// TIA Portal V18 export
FUNCTION_BLOCK "HMI"   // FB20, LAD
TITLE = HMI
{ S7_Optimized_Access := 'TRUE' }
// Bonanza Elect TD Rev0
// Written By Kristopher Gimenez Feb 13,2023
// 
// This block and its associated DB are used for HMI specific actions, interlocks and visualizations.
// stored: AutoNumber false, MemoryReserve 100, SetENOAutomatically false
   VAR
      DHScreen : Array[0..4] of Int;   // Current Info of the Doghouse HMI
      HPUScreen : Array[0..4] of Int;   // Current Info Number of the HPU HMI
      ConsoleScreen : Array[0..4] of Int;   // Current Info Number of the Console HMI
      OscEnable : Bool;   // Oscillator Enable Bit. Set on HMI
      OscAllowEn : Bool;   // Allow Enable from HMI screen.
   END_VAR
   VAR RETAIN
      OscBumpAdj { S7_SetPoint := 'True'} : Real := 20.0;   // Amount the bump position will adjust if increment/decremented. Set on HMI
   END_VAR
   VAR
      OscBumpFwdInc : Bool;   // Used to increase the Fwd Bump by the adjust amount
      OscBumpFwdDec : Bool;   // Used to dec the Fwd Bump by the adjust amount
      OscBumpReactive : Bool;   // Used to trigger Reactive Bump. Always FWD
      OscBumpRevInc : Bool;   // Used to increase the RevBump by the adjust amount
      OscBumpRevDec : Bool;   // Used to dec the Rev Bump by the adjust amount
      OscBumpFwd : Bool;   // Bit used to increase the Home position
      OscBumpRev : Bool;   // Bit used to decrease the home position
   END_VAR
   VAR RETAIN
      OscBumpFwdDeg : Real;   // Amount of Degrees to Bump Forward
      OscBumpRevDeg : Real;   // Amount of Degress to Bump in Rev
   END_VAR
   VAR
      OscHoldButton : Bool;   // Bit used to change color of Button On HMI
      OscHold : Bool;   // Bit used to hold Osc at current position.
      OscBumpFwdButton : Bool;
      OscBumpRevButton : Bool;
      OscBumpFwdRevButtonEn : Bool;
      OscHomeRelDeg : Real;   // Relative Oscillator Home position in degrees.
   END_VAR
   VAR RETAIN
      OscP1FwdMinmA { S7_SetPoint := 'True'} : Real := 200.0;   // Min mA output for Osc FWD on P1
      OscP1FwdMaxmA { S7_SetPoint := 'True'} : Real := 600.0;   // Max mA output for Osc FWD on P1
      OscP1RevMinmA { S7_SetPoint := 'True'} : Real := 200.0;   // Min mA output for Osc Rev on P1
      OscP1RevMaxmA { S7_SetPoint := 'True'} : Real := 600.0;   // Max mA output for Osc Rev on P1
      OscP1HoldmA { S7_SetPoint := 'True'} : Real := 300.0;   // mA Setting to hold position while oscillating
      OscP2FwdMinmA { S7_SetPoint := 'True'} : Real := 200.0;   // Min mA output for Osc FWD on P2
      OscP2FwdMaxmA { S7_SetPoint := 'True'} : Real := 600.0;   // Max mA output for Osc FWD on P2
      OscP2RevMinmA { S7_SetPoint := 'True'} : Real := 200.0;   // Min mA output for Osc Rev on P2
      OscP2RevMaxmA { S7_SetPoint := 'True'} : Real := 600.0;   // Max mA output for Osc Rev on P2
      OscP2HoldmA { S7_SetPoint := 'True'} : Real := 300.0;   // mA Setting to hold position while oscillating
   END_VAR
   VAR
      OscPosZero : Bool;   // Bit used toset the current rotary position as zero degrees and reset Home.
   END_VAR
   VAR RETAIN
      OscSlewRiseFast { S7_SetPoint := 'True'} : Real := 100.0;   // Rising Slew Rate mA/sec for Flow, fast reaction
      OscSlewRiseSlow { S7_SetPoint := 'True'} : Real := 10.0;   // Rising Slew Rate mA/sec on Flow, slow reaction
      OscSlewFallFast { S7_SetPoint := 'True'} : Real := 100.0;   // Falling Slew Rate mA/sec for Flow, fast reaction
      OscSlewFallSlow { S7_SetPoint := 'True'} : Real := 10.0;   // Falling Slew Rate mA/sec on Flow, slow reaction
      OscSpeedTHper { S7_SetPoint := 'True'} : Real := 75.0;   // Speed threshold percent to determine fast or slow slew rates
      OscSpeedHoldper { S7_SetPoint := 'True'} : Real := 95.0;   // Speed threshold percent to where control is held.
      OscSpeedFwdRPM { S7_SetPoint := 'True'} : Real := 15.0;   // Osc FWD speed setpoint. Set on HMI
      OscSpeedRevRPM { S7_SetPoint := 'True'} : Real := 15.0;   // Osc Rev speed setpoint Set on HMI
   END_VAR
   VAR
      OscSpeedFwdZone1 : Real;   // Calc value base on Input and TH percent. Below this speed setpoint - fast ramp up to the speed
      OscSpeedFwdZone2 : Real;   // Calc value base on Input and TH percent, Between Set 1 and Set 2 - Slow ramp up to speed
      OscSpeedFwdZone3 : Real;   // Calc value base on Input and TH percent,Between Set 2 and Set 3 - Maintina Speed
      OscSpeedFwdZone4 : Real;   // Calc value base on Input and TH percent,Between Set 3 and 4 - Slow Ramp Down. Above this speed Fast ramp down
      OscSpeedRevZone1 : Real;   // Calc value base on Input and TH percent. Below this speed setpoint - fast ramp up to the speed
      OscSpeedRevZone2 : Real;   // Calc value base on Input and TH percent, Between Set 1 and Set 2 - Slow ramp up to speed
      OscSpeedRevZone3 : Real;   // Calc value base on Input and TH percent,Between Set 2 and Set 3 - Maintina Speed
      OscSpeedRevZone4 : Real;   // Calc value base on Input and TH percent,Between Set 3 and 4 - Slow Ramp Down. Above this speed Fast ramp down
      OscStart : Bool;   // Bit used to start Oscillating
      OscStartButton : Bool;   // Bit used to change color of Button On HMI
      OscStop : Bool;   // Bit used to Stop Oscillating or Holding
      OscStopButton : Bool;   // Bit used to change color of Button On HMI
   END_VAR
   VAR RETAIN
      OscTorqAdj { S7_SetPoint := 'True'} : Real := 500.0;   // Amount the torq will adjust if increment/decremented. Set on HMI
      OscTorqFwdFtLbs : Real := 5000.0;   // Osc fwd torq setpoint
   END_VAR
   VAR
      OscTorqFwdInc : Bool;   // Increment Torq Fwd
      OscTorqFwdDec : Bool;   // Decrement Torq Fwd
      OscTorqRevInc : Bool;   // Increment Torq Rev
   END_VAR
   VAR RETAIN
      OscTorqRevFtLbs : Real := 5000.0;   // Osc Rev Torq Setpoint
   END_VAR
   VAR
      OscTorqRevDec : Bool;   // Decrement Torq REv
      OscTorqSetPSI : Real;
   END_VAR
   VAR RETAIN
      OscTurnAdj { S7_SetPoint := 'True'} : Real := 0.25;   // Amount the turns will adjust if increment/decremented. Set on HMI
      OscTurnFwd : Real := 1.0;   // Osc Fwd Turns
   END_VAR
   VAR
      OscTurnFwdInc : Bool;   // Increment Turns Fwd
      OscTurnFwdDec : Bool;   // Decrement Turns Fwd
   END_VAR
   VAR RETAIN
      OscTurnRev : Real := 1.0;   // Osc Rev Turns
   END_VAR
   VAR
      OscTurnRevInc : Bool;   // Increment Turns Rev
      OscTurnRevDec : Bool;   // Decrement Turns Rev
      OscTorqFwdLowLimFtlbs : Real;   // Forward torq lower limit based on input and settings
      OscTorqFwdHighLimFtLbs : Real;   // Forward torq high limit based on input and settings
      OscTorqRevLowLimFtlbs : Real;   // Reverse torq lower limit based on input and settings
      OscTorqRevHighLimFtLbs : Real;   // Reverse torq high limit based on input and settings
      OscHomeLowRelDeg : Real;   // Rel Home Position minus 1 count range
      OscHomeLow2RelDeg : Real;   // Rel Home Position minus 2 count range
      OscHomeHighRelDeg : Real;   // Rel Home Position plus 1 count range
      OscHomeHigh2RelDeg : Real;   // Rel Home Position plus 2 count range
      OscPosDeg : Real;   // Degrees of from Home position
      SpareVolts : Real := 0.0;   // Dummy spare Output value used for display
      Spare4MA : Real := 4.0;   // Dummy spare Output value 4ma
      LampTest : Bool;   // Bit used to trigger Console lamp test from HMI
      LampTestLamp_TP { S7_SetPoint := 'True'} : TP_TIME;
      LampTestHorn_TP { S7_SetPoint := 'True'} : TP_TIME;
      ScreenNameInvis { S7_SetPoint := 'True'} : Bool;   // Used to Turn off Screen Name
      ScreenBypassVis : Bool;
      ScreenLampTestVis : Bool;
      HornSilence_TOF { S7_SetPoint := 'True'} : TOF_TIME;
      HornSilenceReset { S7_SetPoint := 'True'} : Bool;   // Horn Silence Bit set on HMI
      Alarms1 : Int;
      Alarms2 : Int;
      Warnings1 : Int;
      Alarms1_To_Unified : Array[0..15] of Bool;
      Alarms2_To_Unified : Array[0..15] of Bool;
      Warnings1_To_Unified : Array[0..15] of Bool;
   END_VAR
   VAR_TEMP
      TempReal : Real;
   END_VAR
   VAR_TEMP   // added for the SCL form of the ladder/FBD networks
      _w1 : Bool;
   END_VAR
BEGIN

REGION Network 1: Oscillator Enable
   // Allow Enable Osciallor Set from HMI if  in Drill, throttle pot set to min and TD stopped, low speed. 
   // HMI Used to Set Enable
   // Reset if Interlocks not met
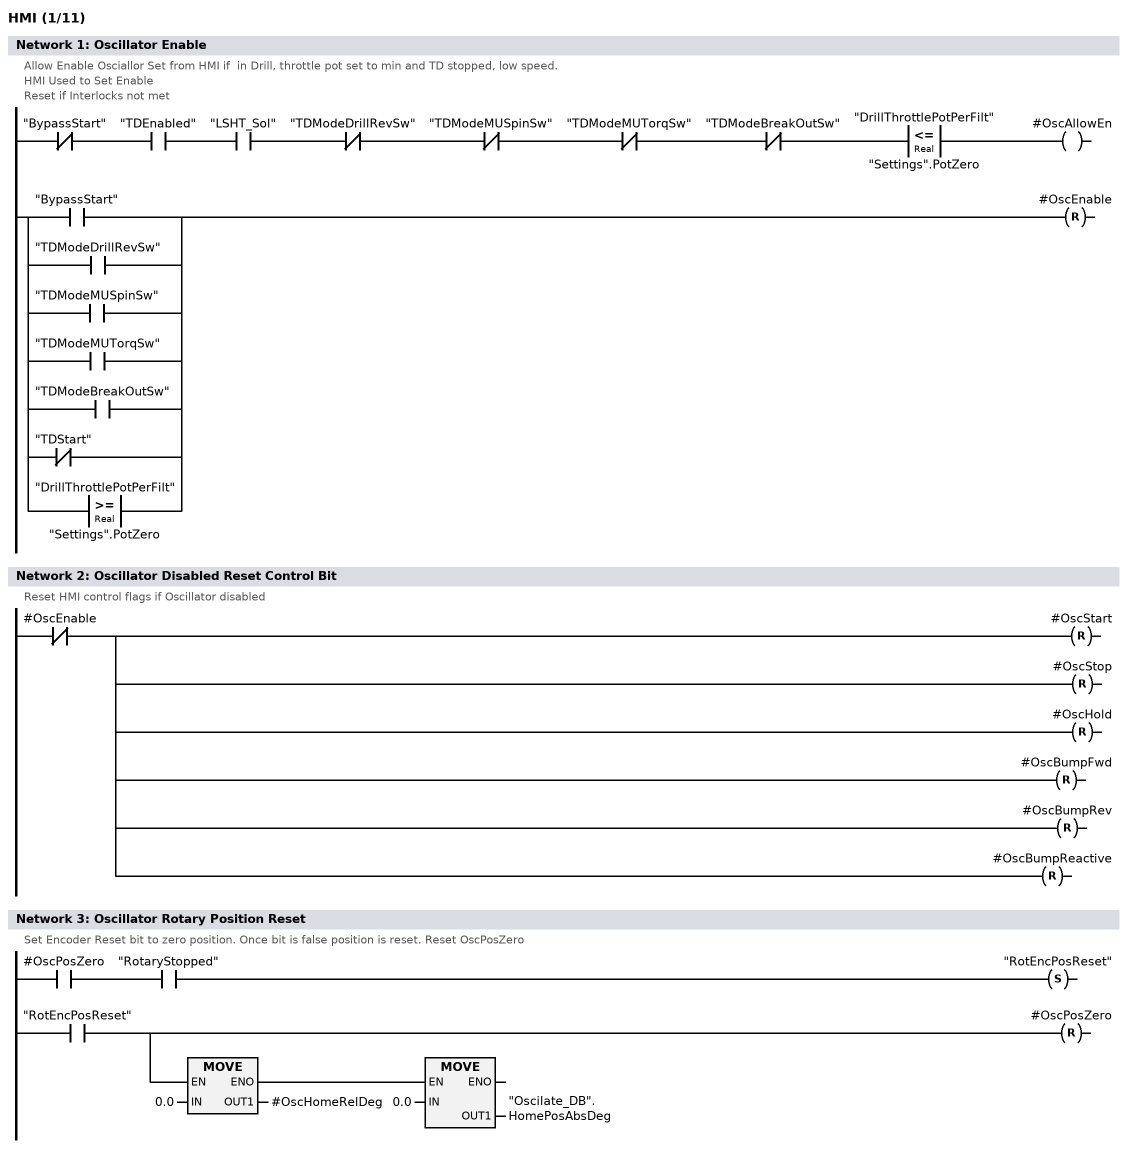
   RUNG wire#powerrail
      I_Contact( "BypassStart" )
      Contact( "TDEnabled" )
      Contact( "LSHT_Sol" )
      I_Contact( "TDModeDrillRevSw" )
      I_Contact( "TDModeMUSpinSw" )
      I_Contact( "TDModeMUTorqSw" )
      I_Contact( "TDModeBreakOutSw" )
      { S7_Templates := "SrcType := Real" } LE_Contact(in1 := "DrillThrottlePotPerFilt", in2 := "Settings".PotZero)
      Coil( #OscAllowEn )
   END_RUNG
   RUNG wire#powerrail
      Contact( "BypassStart" )
      wire#w1
      R_Coil( #OscEnable )
   END_RUNG
   RUNG wire#powerrail
      Contact( "TDModeDrillRevSw" )
   END_RUNG wire#w1
   RUNG wire#powerrail
      Contact( "TDModeMUSpinSw" )
   END_RUNG wire#w1
   RUNG wire#powerrail
      Contact( "TDModeMUTorqSw" )
   END_RUNG wire#w1
   RUNG wire#powerrail
      Contact( "TDModeBreakOutSw" )
   END_RUNG wire#w1
   RUNG wire#powerrail
      I_Contact( "TDStart" )
   END_RUNG wire#w1
   RUNG wire#powerrail
      { S7_Templates := "SrcType := Real" } GE_Contact(in1 := "DrillThrottlePotPerFilt", in2 := "Settings".PotZero)
   END_RUNG wire#w1
   // the same network as SCL:
   #OscAllowEn := NOT "BypassStart" AND "TDEnabled" AND "LSHT_Sol" AND NOT "TDModeDrillRevSw" AND NOT "TDModeMUSpinSw" AND NOT "TDModeMUTorqSw" AND NOT "TDModeBreakOutSw" AND ("DrillThrottlePotPerFilt" <= "Settings".PotZero);
   IF "BypassStart" OR "TDModeDrillRevSw" OR "TDModeMUSpinSw" OR "TDModeMUTorqSw" OR "TDModeBreakOutSw" OR NOT "TDStart" OR ("DrillThrottlePotPerFilt" >= "Settings".PotZero) THEN
       #OscEnable := FALSE;
   END_IF;
END_REGION

REGION Network 2: Oscillator Disabled Reset Control Bit
   // Reset HMI control flags if Oscillator disabled
   RUNG wire#powerrail
      I_Contact( #OscEnable )
      wire#w1
      R_Coil( #OscStart )
   END_RUNG
   RUNG wire#w1
      R_Coil( #OscStop )
   END_RUNG
   RUNG wire#w1
      R_Coil( #OscHold )
   END_RUNG
   RUNG wire#w1
      R_Coil( #OscBumpFwd )
   END_RUNG
   RUNG wire#w1
      R_Coil( #OscBumpRev )
   END_RUNG
   RUNG wire#w1
      R_Coil( #OscBumpReactive )
   END_RUNG
   // the same network as SCL:
   IF NOT #OscEnable THEN
       #OscStart := FALSE;
       #OscStop := FALSE;
       #OscHold := FALSE;
       #OscBumpFwd := FALSE;
       #OscBumpRev := FALSE;
       #OscBumpReactive := FALSE;
   END_IF;
END_REGION

REGION Network 3: Oscillator Rotary Position Reset
   // Set Encoder Reset bit to zero position. Once bit is false position is reset. Reset OscPosZero
   RUNG wire#powerrail
      Contact( #OscPosZero )
      Contact( "RotaryStopped" )
      S_Coil( "RotEncPosReset" )
   END_RUNG
   RUNG wire#powerrail
      Contact( "RotEncPosReset" )
      wire#w1
      R_Coil( #OscPosZero )
   END_RUNG
   RUNG wire#w1
      Move(in := 0.0, out1 => #OscHomeRelDeg)
      Move(in := 0.0, out1 => "Oscilate_DB".HomePosAbsDeg)
   END_RUNG
   // the same network as SCL:
   IF #OscPosZero AND "RotaryStopped" THEN "RotEncPosReset" := TRUE; END_IF;
   IF "RotEncPosReset" THEN
       #OscPosZero := FALSE;
       #OscHomeRelDeg := 0.0;
       "Oscilate_DB".HomePosAbsDeg := 0.0;
   END_IF;
END_REGION

REGION Network 4: Oscillator Position
   // Determine Oscillation position based on home position and actual absolute position
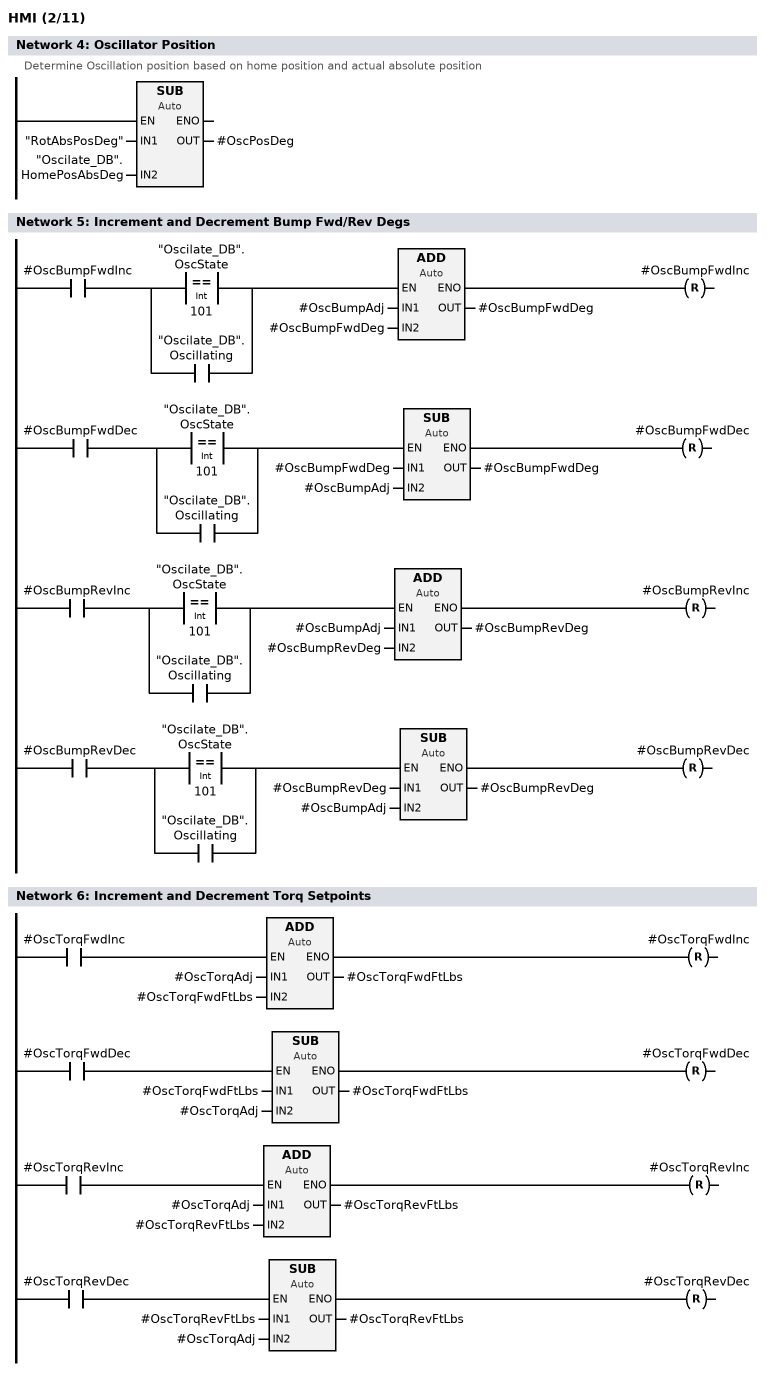
   RUNG wire#powerrail
      Sub(in1 := "RotAbsPosDeg", in2 := "Oscilate_DB".HomePosAbsDeg, out => #OscPosDeg)
   END_RUNG
   // the same network as SCL:
   #OscPosDeg := "RotAbsPosDeg" - "Oscilate_DB".HomePosAbsDeg;
END_REGION

REGION Network 5: Increment and Decrement Bump Fwd/Rev Degs
   RUNG wire#powerrail
      Contact( #OscBumpFwdInc )
      wire#w1
      { S7_Templates := "SrcType := Int" } EQ_Contact(in1 := "Oscilate_DB".OscState, in2 := 101)
      wire#w2
      Add(in1 := #OscBumpAdj, in2 := #OscBumpFwdDeg, out => #OscBumpFwdDeg)
      R_Coil( #OscBumpFwdInc )
   END_RUNG
   RUNG wire#w1
      Contact( "Oscilate_DB".Oscillating )
   END_RUNG wire#w2
   RUNG wire#powerrail
      Contact( #OscBumpFwdDec )
      wire#w3
      { S7_Templates := "SrcType := Int" } EQ_Contact(in1 := "Oscilate_DB".OscState, in2 := 101)
      wire#w4
      Sub(in1 := #OscBumpFwdDeg, in2 := #OscBumpAdj, out => #OscBumpFwdDeg)
      R_Coil( #OscBumpFwdDec )
   END_RUNG
   RUNG wire#w3
      Contact( "Oscilate_DB".Oscillating )
   END_RUNG wire#w4
   RUNG wire#powerrail
      Contact( #OscBumpRevInc )
      wire#w5
      { S7_Templates := "SrcType := Int" } EQ_Contact(in1 := "Oscilate_DB".OscState, in2 := 101)
      wire#w6
      Add(in1 := #OscBumpAdj, in2 := #OscBumpRevDeg, out => #OscBumpRevDeg)
      R_Coil( #OscBumpRevInc )
   END_RUNG
   RUNG wire#w5
      Contact( "Oscilate_DB".Oscillating )
   END_RUNG wire#w6
   RUNG wire#powerrail
      Contact( #OscBumpRevDec )
      wire#w7
      { S7_Templates := "SrcType := Int" } EQ_Contact(in1 := "Oscilate_DB".OscState, in2 := 101)
      wire#w8
      Sub(in1 := #OscBumpRevDeg, in2 := #OscBumpAdj, out => #OscBumpRevDeg)
      R_Coil( #OscBumpRevDec )
   END_RUNG
   RUNG wire#w7
      Contact( "Oscilate_DB".Oscillating )
   END_RUNG wire#w8
   // the same network as SCL:
   IF #OscBumpFwdInc AND (("Oscilate_DB".OscState = 101) OR "Oscilate_DB".Oscillating) THEN
       #OscBumpFwdDeg := #OscBumpAdj + #OscBumpFwdDeg;
       #OscBumpFwdInc := FALSE;
   END_IF;
   IF #OscBumpFwdDec AND (("Oscilate_DB".OscState = 101) OR "Oscilate_DB".Oscillating) THEN
       #OscBumpFwdDeg := #OscBumpFwdDeg - #OscBumpAdj;
       #OscBumpFwdDec := FALSE;
   END_IF;
   IF #OscBumpRevInc AND (("Oscilate_DB".OscState = 101) OR "Oscilate_DB".Oscillating) THEN
       #OscBumpRevDeg := #OscBumpAdj + #OscBumpRevDeg;
       #OscBumpRevInc := FALSE;
   END_IF;
   IF #OscBumpRevDec AND (("Oscilate_DB".OscState = 101) OR "Oscilate_DB".Oscillating) THEN
       #OscBumpRevDeg := #OscBumpRevDeg - #OscBumpAdj;
       #OscBumpRevDec := FALSE;
   END_IF;
END_REGION

REGION Network 6: Increment and Decrement Torq Setpoints
   RUNG wire#powerrail
      Contact( #OscTorqFwdInc )
      Add(in1 := #OscTorqAdj, in2 := #OscTorqFwdFtLbs, out => #OscTorqFwdFtLbs)
      R_Coil( #OscTorqFwdInc )
   END_RUNG
   RUNG wire#powerrail
      Contact( #OscTorqFwdDec )
      Sub(in1 := #OscTorqFwdFtLbs, in2 := #OscTorqAdj, out => #OscTorqFwdFtLbs)
      R_Coil( #OscTorqFwdDec )
   END_RUNG
   RUNG wire#powerrail
      Contact( #OscTorqRevInc )
      Add(in1 := #OscTorqAdj, in2 := #OscTorqRevFtLbs, out => #OscTorqRevFtLbs)
      R_Coil( #OscTorqRevInc )
   END_RUNG
   RUNG wire#powerrail
      Contact( #OscTorqRevDec )
      Sub(in1 := #OscTorqRevFtLbs, in2 := #OscTorqAdj, out => #OscTorqRevFtLbs)
      R_Coil( #OscTorqRevDec )
   END_RUNG
   // the same network as SCL:
   IF #OscTorqFwdInc THEN
       #OscTorqFwdFtLbs := #OscTorqAdj + #OscTorqFwdFtLbs;
       #OscTorqFwdInc := FALSE;
   END_IF;
   IF #OscTorqFwdDec THEN
       #OscTorqFwdFtLbs := #OscTorqFwdFtLbs - #OscTorqAdj;
       #OscTorqFwdDec := FALSE;
   END_IF;
   IF #OscTorqRevInc THEN
       #OscTorqRevFtLbs := #OscTorqAdj + #OscTorqRevFtLbs;
       #OscTorqRevInc := FALSE;
   END_IF;
   IF #OscTorqRevDec THEN
       #OscTorqRevFtLbs := #OscTorqRevFtLbs - #OscTorqAdj;
       #OscTorqRevDec := FALSE;
   END_IF;
END_REGION

REGION Network 7: Increment and Decrement Turns
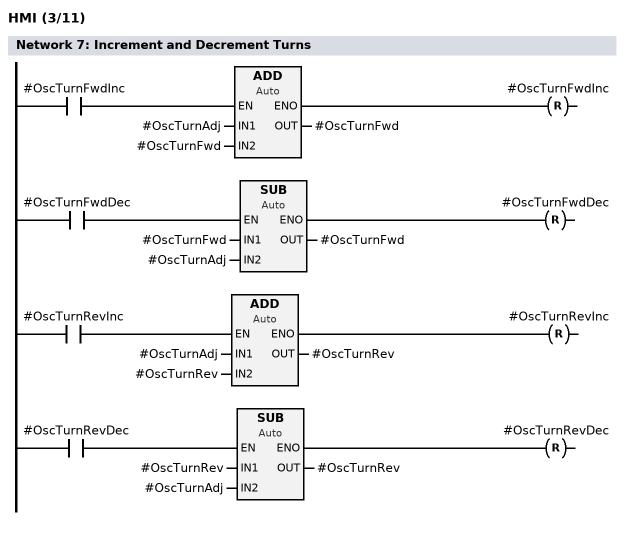
   RUNG wire#powerrail
      Contact( #OscTurnFwdInc )
      Add(in1 := #OscTurnAdj, in2 := #OscTurnFwd, out => #OscTurnFwd)
      R_Coil( #OscTurnFwdInc )
   END_RUNG
   RUNG wire#powerrail
      Contact( #OscTurnFwdDec )
      Sub(in1 := #OscTurnFwd, in2 := #OscTurnAdj, out => #OscTurnFwd)
      R_Coil( #OscTurnFwdDec )
   END_RUNG
   RUNG wire#powerrail
      Contact( #OscTurnRevInc )
      Add(in1 := #OscTurnAdj, in2 := #OscTurnRev, out => #OscTurnRev)
      R_Coil( #OscTurnRevInc )
   END_RUNG
   RUNG wire#powerrail
      Contact( #OscTurnRevDec )
      Sub(in1 := #OscTurnRev, in2 := #OscTurnAdj, out => #OscTurnRev)
      R_Coil( #OscTurnRevDec )
   END_RUNG
   // the same network as SCL:
   IF #OscTurnFwdInc THEN
       #OscTurnFwd := #OscTurnAdj + #OscTurnFwd;
       #OscTurnFwdInc := FALSE;
   END_IF;
   IF #OscTurnFwdDec THEN
       #OscTurnFwd := #OscTurnFwd - #OscTurnAdj;
       #OscTurnFwdDec := FALSE;
   END_IF;
   IF #OscTurnRevInc THEN
       #OscTurnRev := #OscTurnAdj + #OscTurnRev;
       #OscTurnRevInc := FALSE;
   END_IF;
   IF #OscTurnRevDec THEN
       #OscTurnRev := #OscTurnRev - #OscTurnAdj;
       #OscTurnRevDec := FALSE;
   END_IF;
END_REGION

REGION Network 8: Oscillator Input Limits Checks
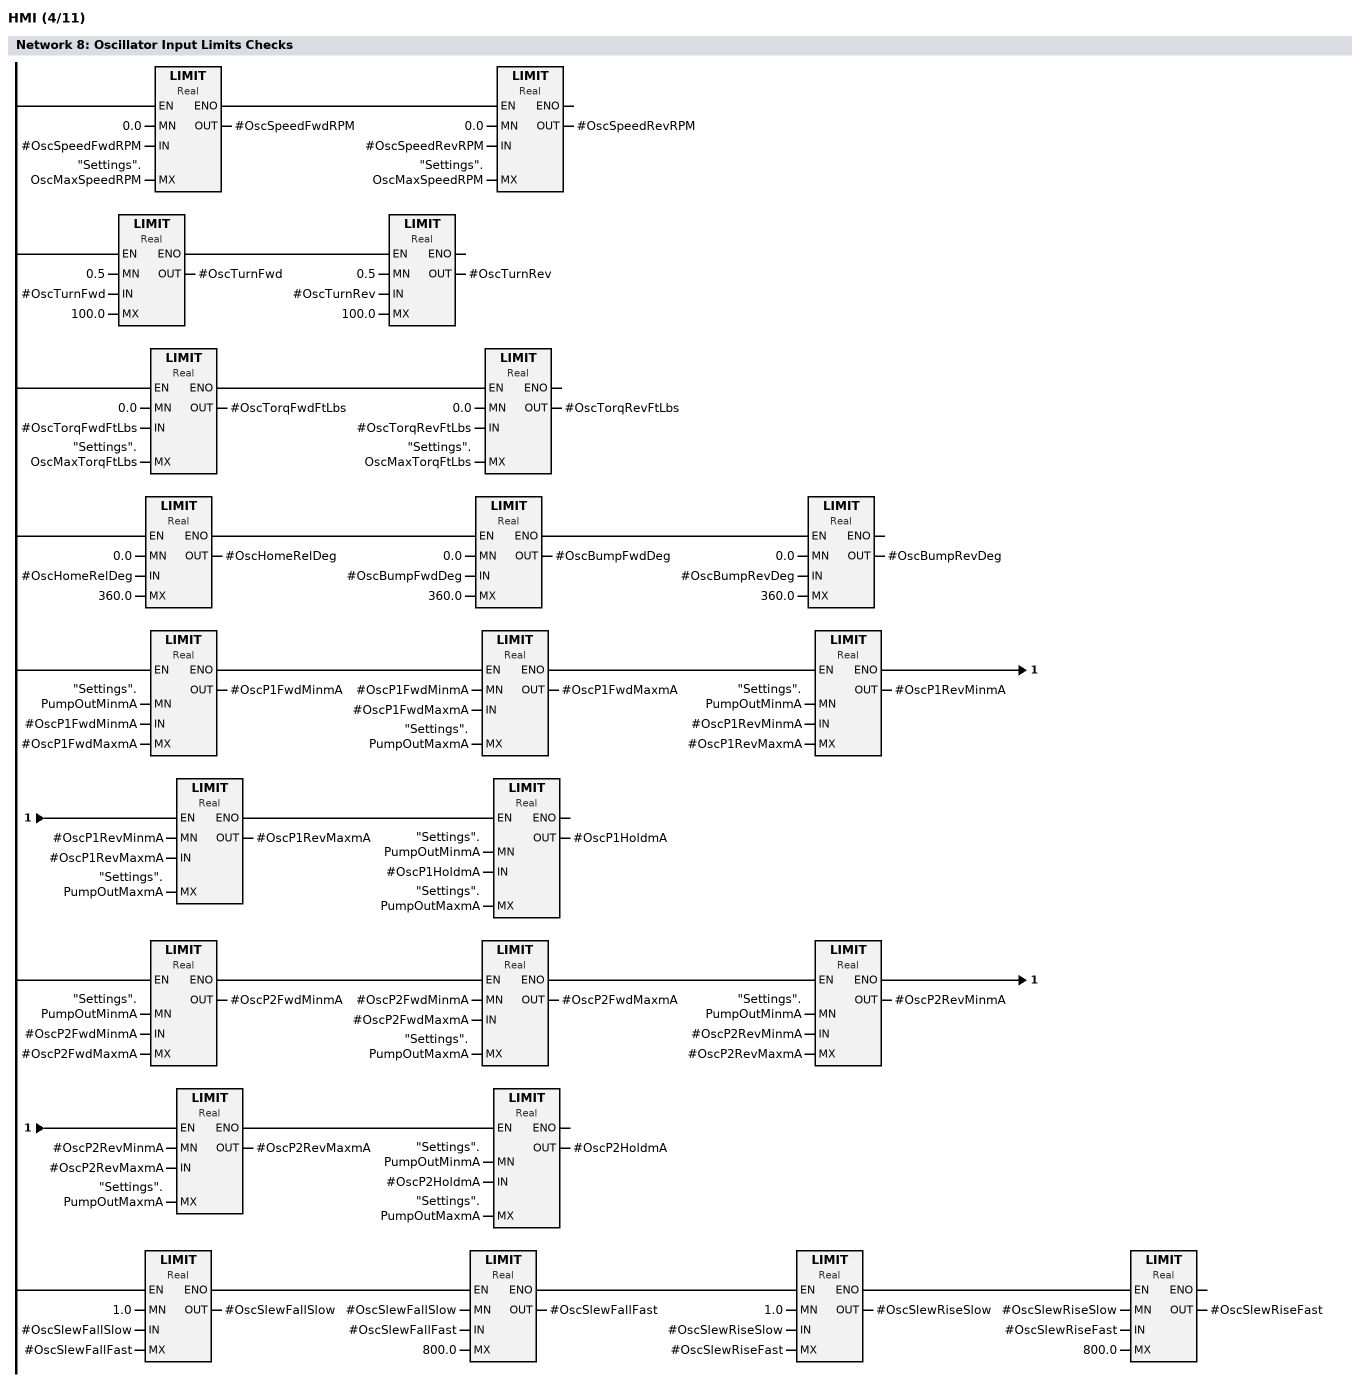
   RUNG wire#powerrail
      { S7_Templates := "value_type := Real" } Limit(mn := 0.0, in := #OscSpeedFwdRPM, mx := "Settings".OscMaxSpeedRPM, out => #OscSpeedFwdRPM)
      { S7_Templates := "value_type := Real" } Limit(mn := 0.0, in := #OscSpeedRevRPM, mx := "Settings".OscMaxSpeedRPM, out => #OscSpeedRevRPM)
   END_RUNG
   RUNG wire#powerrail
      { S7_Templates := "value_type := Real" } Limit(mn := 0.5, in := #OscTurnFwd, mx := 100.0, out => #OscTurnFwd)
      { S7_Templates := "value_type := Real" } Limit(mn := 0.5, in := #OscTurnRev, mx := 100.0, out => #OscTurnRev)
   END_RUNG
   RUNG wire#powerrail
      { S7_Templates := "value_type := Real" } Limit(mn := 0.0, in := #OscTorqFwdFtLbs, mx := "Settings".OscMaxTorqFtLbs, out => #OscTorqFwdFtLbs)
      { S7_Templates := "value_type := Real" } Limit(mn := 0.0, in := #OscTorqRevFtLbs, mx := "Settings".OscMaxTorqFtLbs, out => #OscTorqRevFtLbs)
   END_RUNG
   RUNG wire#powerrail
      { S7_Templates := "value_type := Real" } Limit(mn := 0.0, in := #OscHomeRelDeg, mx := 360.0, out => #OscHomeRelDeg)
      { S7_Templates := "value_type := Real" } Limit(mn := 0.0, in := #OscBumpFwdDeg, mx := 360.0, out => #OscBumpFwdDeg)
      { S7_Templates := "value_type := Real" } Limit(mn := 0.0, in := #OscBumpRevDeg, mx := 360.0, out => #OscBumpRevDeg)
   END_RUNG
   RUNG wire#powerrail
      { S7_Templates := "value_type := Real" } Limit(mn := "Settings".PumpOutMinmA, in := #OscP1FwdMinmA, mx := #OscP1FwdMaxmA, out => #OscP1FwdMinmA)
      { S7_Templates := "value_type := Real" } Limit(mn := #OscP1FwdMinmA, in := #OscP1FwdMaxmA, mx := "Settings".PumpOutMaxmA, out => #OscP1FwdMaxmA)
      { S7_Templates := "value_type := Real" } Limit(mn := "Settings".PumpOutMinmA, in := #OscP1RevMinmA, mx := #OscP1RevMaxmA, out => #OscP1RevMinmA)
      { S7_Templates := "value_type := Real" } Limit(mn := #OscP1RevMinmA, in := #OscP1RevMaxmA, mx := "Settings".PumpOutMaxmA, out => #OscP1RevMaxmA)
      { S7_Templates := "value_type := Real" } Limit(mn := "Settings".PumpOutMinmA, in := #OscP1HoldmA, mx := "Settings".PumpOutMaxmA, out => #OscP1HoldmA)
   END_RUNG
   RUNG wire#powerrail
      { S7_Templates := "value_type := Real" } Limit(mn := "Settings".PumpOutMinmA, in := #OscP2FwdMinmA, mx := #OscP2FwdMaxmA, out => #OscP2FwdMinmA)
      { S7_Templates := "value_type := Real" } Limit(mn := #OscP2FwdMinmA, in := #OscP2FwdMaxmA, mx := "Settings".PumpOutMaxmA, out => #OscP2FwdMaxmA)
      { S7_Templates := "value_type := Real" } Limit(mn := "Settings".PumpOutMinmA, in := #OscP2RevMinmA, mx := #OscP2RevMaxmA, out => #OscP2RevMinmA)
      { S7_Templates := "value_type := Real" } Limit(mn := #OscP2RevMinmA, in := #OscP2RevMaxmA, mx := "Settings".PumpOutMaxmA, out => #OscP2RevMaxmA)
      { S7_Templates := "value_type := Real" } Limit(mn := "Settings".PumpOutMinmA, in := #OscP2HoldmA, mx := "Settings".PumpOutMaxmA, out => #OscP2HoldmA)
   END_RUNG
   RUNG wire#powerrail
      { S7_Templates := "value_type := Real" } Limit(mn := 1.0, in := #OscSlewFallSlow, mx := #OscSlewFallFast, out => #OscSlewFallSlow)
      { S7_Templates := "value_type := Real" } Limit(mn := #OscSlewFallSlow, in := #OscSlewFallFast, mx := 800.0, out => #OscSlewFallFast)
      { S7_Templates := "value_type := Real" } Limit(mn := 1.0, in := #OscSlewRiseSlow, mx := #OscSlewRiseFast, out => #OscSlewRiseSlow)
      { S7_Templates := "value_type := Real" } Limit(mn := #OscSlewRiseSlow, in := #OscSlewRiseFast, mx := 800.0, out => #OscSlewRiseFast)
   END_RUNG
   // the same network as SCL:
   #OscSpeedFwdRPM := LIMIT(MN := 0.0, IN := #OscSpeedFwdRPM, MX := "Settings".OscMaxSpeedRPM);
   #OscSpeedRevRPM := LIMIT(MN := 0.0, IN := #OscSpeedRevRPM, MX := "Settings".OscMaxSpeedRPM);
   #OscTurnFwd := LIMIT(MN := 0.5, IN := #OscTurnFwd, MX := 100.0);
   #OscTurnRev := LIMIT(MN := 0.5, IN := #OscTurnRev, MX := 100.0);
   #OscTorqFwdFtLbs := LIMIT(MN := 0.0, IN := #OscTorqFwdFtLbs, MX := "Settings".OscMaxTorqFtLbs);
   #OscTorqRevFtLbs := LIMIT(MN := 0.0, IN := #OscTorqRevFtLbs, MX := "Settings".OscMaxTorqFtLbs);
   #OscHomeRelDeg := LIMIT(MN := 0.0, IN := #OscHomeRelDeg, MX := 360.0);
   #OscBumpFwdDeg := LIMIT(MN := 0.0, IN := #OscBumpFwdDeg, MX := 360.0);
   #OscBumpRevDeg := LIMIT(MN := 0.0, IN := #OscBumpRevDeg, MX := 360.0);
   #OscP1FwdMinmA := LIMIT(MN := "Settings".PumpOutMinmA, IN := #OscP1FwdMinmA, MX := #OscP1FwdMaxmA);
   #OscP1FwdMaxmA := LIMIT(MN := #OscP1FwdMinmA, IN := #OscP1FwdMaxmA, MX := "Settings".PumpOutMaxmA);
   #OscP1RevMinmA := LIMIT(MN := "Settings".PumpOutMinmA, IN := #OscP1RevMinmA, MX := #OscP1RevMaxmA);
   #OscP1RevMaxmA := LIMIT(MN := #OscP1RevMinmA, IN := #OscP1RevMaxmA, MX := "Settings".PumpOutMaxmA);
   #OscP1HoldmA := LIMIT(MN := "Settings".PumpOutMinmA, IN := #OscP1HoldmA, MX := "Settings".PumpOutMaxmA);
   #OscP2FwdMinmA := LIMIT(MN := "Settings".PumpOutMinmA, IN := #OscP2FwdMinmA, MX := #OscP2FwdMaxmA);
   #OscP2FwdMaxmA := LIMIT(MN := #OscP2FwdMinmA, IN := #OscP2FwdMaxmA, MX := "Settings".PumpOutMaxmA);
   #OscP2RevMinmA := LIMIT(MN := "Settings".PumpOutMinmA, IN := #OscP2RevMinmA, MX := #OscP2RevMaxmA);
   #OscP2RevMaxmA := LIMIT(MN := #OscP2RevMinmA, IN := #OscP2RevMaxmA, MX := "Settings".PumpOutMaxmA);
   #OscP2HoldmA := LIMIT(MN := "Settings".PumpOutMinmA, IN := #OscP2HoldmA, MX := "Settings".PumpOutMaxmA);
   #OscSlewFallSlow := LIMIT(MN := 1.0, IN := #OscSlewFallSlow, MX := #OscSlewFallFast);
   #OscSlewFallFast := LIMIT(MN := #OscSlewFallSlow, IN := #OscSlewFallFast, MX := 800.0);
   #OscSlewRiseSlow := LIMIT(MN := 1.0, IN := #OscSlewRiseSlow, MX := #OscSlewRiseFast);
   #OscSlewRiseFast := LIMIT(MN := #OscSlewRiseSlow, IN := #OscSlewRiseFast, MX := 800.0);
END_REGION

REGION Network 9: Calculate Torq Setpoint
   // Only Fwd Torq is used to set torq
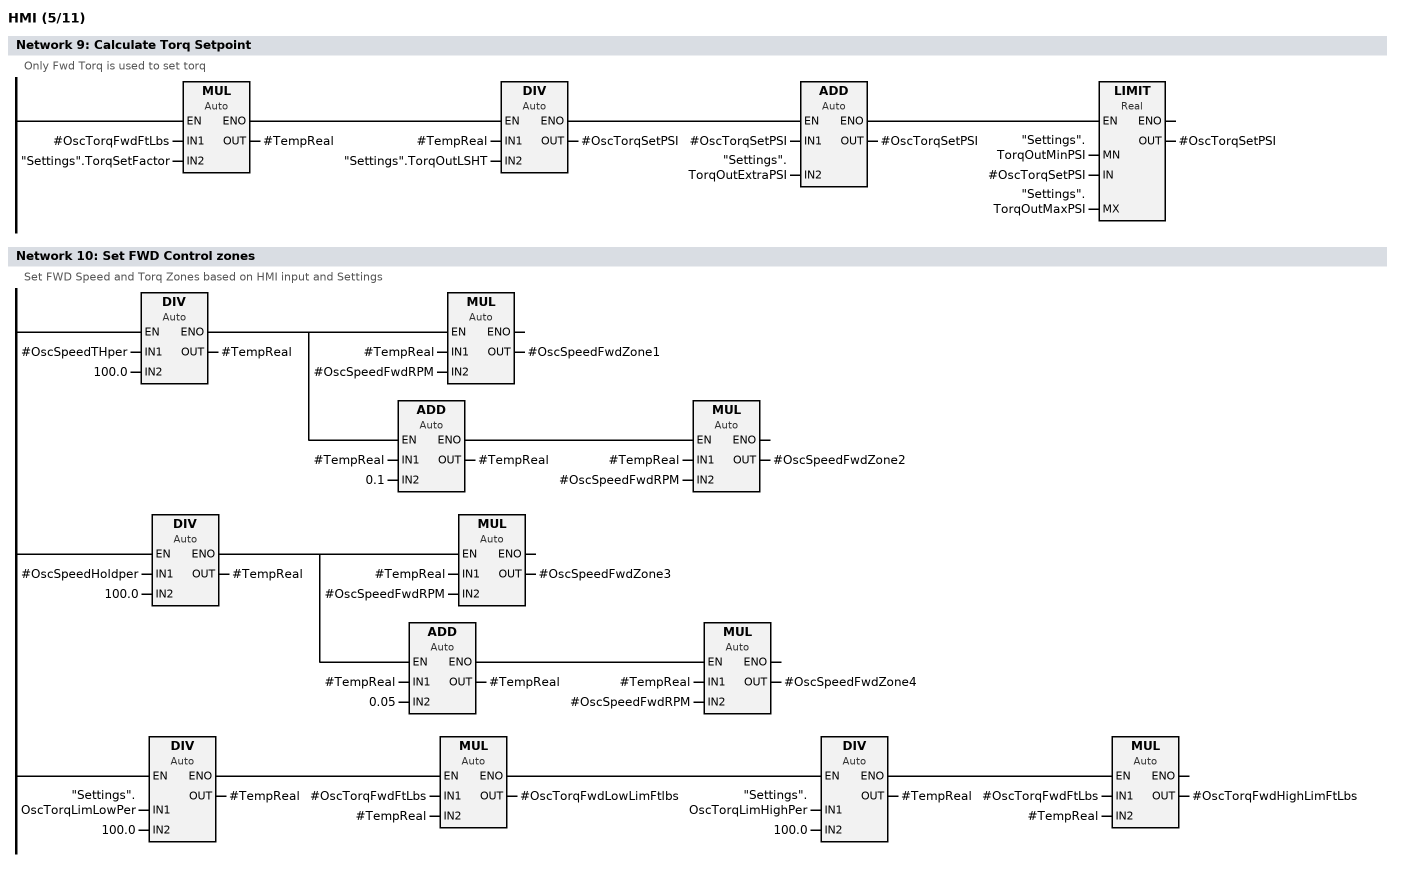
   RUNG wire#powerrail
      Mul(in1 := #OscTorqFwdFtLbs, in2 := "Settings".TorqSetFactor, out => #TempReal)
      Div(in1 := #TempReal, in2 := "Settings".TorqOutLSHT, out => #OscTorqSetPSI)
      Add(in1 := #OscTorqSetPSI, in2 := "Settings".TorqOutExtraPSI, out => #OscTorqSetPSI)
      { S7_Templates := "value_type := Real" } Limit(mn := "Settings".TorqOutMinPSI, in := #OscTorqSetPSI, mx := "Settings".TorqOutMaxPSI, out => #OscTorqSetPSI)
   END_RUNG
   // the same network as SCL:
   #TempReal := #OscTorqFwdFtLbs * "Settings".TorqSetFactor;
   #OscTorqSetPSI := #TempReal / "Settings".TorqOutLSHT;
   #OscTorqSetPSI := #OscTorqSetPSI + "Settings".TorqOutExtraPSI;
   #OscTorqSetPSI := LIMIT(MN := "Settings".TorqOutMinPSI, IN := #OscTorqSetPSI, MX := "Settings".TorqOutMaxPSI);
END_REGION

REGION Network 10: Set FWD Control zones
   // Set FWD Speed and Torq Zones based on HMI input and Settings
   RUNG wire#powerrail
      Div(in1 := #OscSpeedTHper, in2 := 100.0, out => #TempReal)
      wire#w1
      Mul(in1 := #TempReal, in2 := #OscSpeedFwdRPM, out => #OscSpeedFwdZone1)
   END_RUNG
   RUNG wire#w1
      Add(in1 := #TempReal, in2 := 0.1, out => #TempReal)
      Mul(in1 := #TempReal, in2 := #OscSpeedFwdRPM, out => #OscSpeedFwdZone2)
   END_RUNG
   RUNG wire#powerrail
      Div(in1 := #OscSpeedHoldper, in2 := 100.0, out => #TempReal)
      wire#w2
      Mul(in1 := #TempReal, in2 := #OscSpeedFwdRPM, out => #OscSpeedFwdZone3)
   END_RUNG
   RUNG wire#w2
      Add(in1 := #TempReal, in2 := 0.05, out => #TempReal)
      Mul(in1 := #TempReal, in2 := #OscSpeedFwdRPM, out => #OscSpeedFwdZone4)
   END_RUNG
   RUNG wire#powerrail
      Div(in1 := "Settings".OscTorqLimLowPer, in2 := 100.0, out => #TempReal)
      Mul(in1 := #OscTorqFwdFtLbs, in2 := #TempReal, out => #OscTorqFwdLowLimFtlbs)
      Div(in1 := "Settings".OscTorqLimHighPer, in2 := 100.0, out => #TempReal)
      Mul(in1 := #OscTorqFwdFtLbs, in2 := #TempReal, out => #OscTorqFwdHighLimFtLbs)
   END_RUNG
   // the same network as SCL:
   #TempReal := #OscSpeedTHper / 100.0;
   #OscSpeedFwdZone1 := #TempReal * #OscSpeedFwdRPM;
   #TempReal := #TempReal + 0.1;
   #OscSpeedFwdZone2 := #TempReal * #OscSpeedFwdRPM;
   #TempReal := #OscSpeedHoldper / 100.0;
   #OscSpeedFwdZone3 := #TempReal * #OscSpeedFwdRPM;
   #TempReal := #TempReal + 0.05;
   #OscSpeedFwdZone4 := #TempReal * #OscSpeedFwdRPM;
   #TempReal := "Settings".OscTorqLimLowPer / 100.0;
   #OscTorqFwdLowLimFtlbs := #OscTorqFwdFtLbs * #TempReal;
   #TempReal := "Settings".OscTorqLimHighPer / 100.0;
   #OscTorqFwdHighLimFtLbs := #OscTorqFwdFtLbs * #TempReal;
END_REGION

REGION Network 11: Set Rev Controls zones
   // Set Rev Speed and Torq Zones based on HMI input and Settings
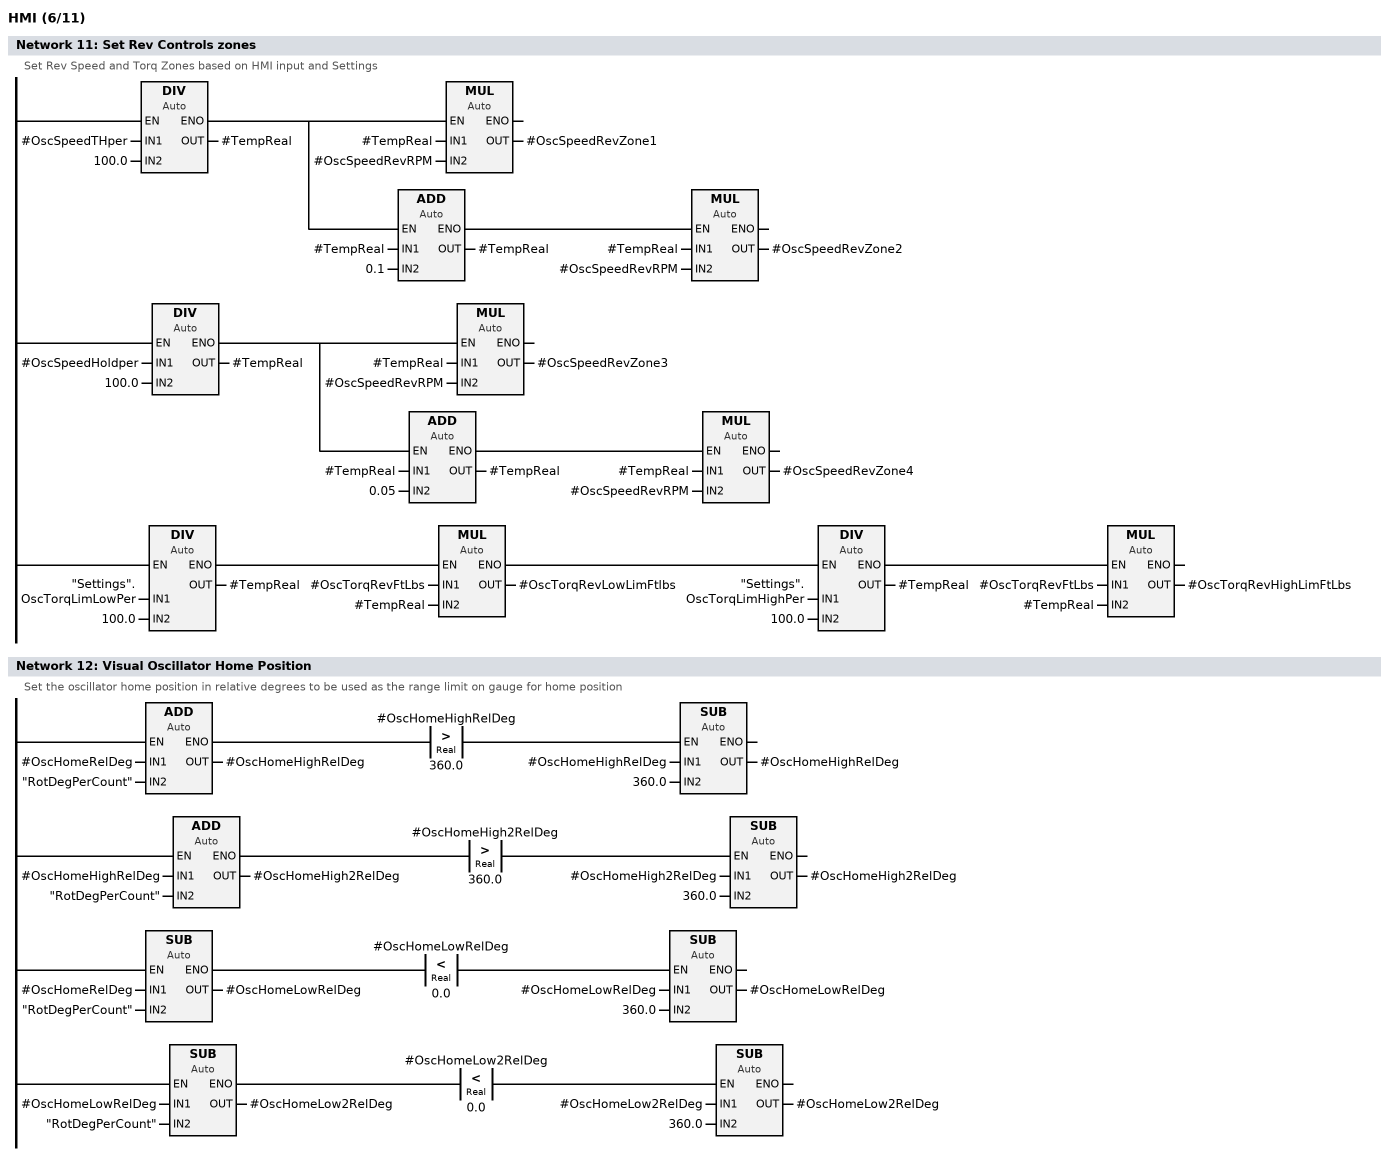
   RUNG wire#powerrail
      Div(in1 := #OscSpeedTHper, in2 := 100.0, out => #TempReal)
      wire#w1
      Mul(in1 := #TempReal, in2 := #OscSpeedRevRPM, out => #OscSpeedRevZone1)
   END_RUNG
   RUNG wire#w1
      Add(in1 := #TempReal, in2 := 0.1, out => #TempReal)
      Mul(in1 := #TempReal, in2 := #OscSpeedRevRPM, out => #OscSpeedRevZone2)
   END_RUNG
   RUNG wire#powerrail
      Div(in1 := #OscSpeedHoldper, in2 := 100.0, out => #TempReal)
      wire#w2
      Mul(in1 := #TempReal, in2 := #OscSpeedRevRPM, out => #OscSpeedRevZone3)
   END_RUNG
   RUNG wire#w2
      Add(in1 := #TempReal, in2 := 0.05, out => #TempReal)
      Mul(in1 := #TempReal, in2 := #OscSpeedRevRPM, out => #OscSpeedRevZone4)
   END_RUNG
   RUNG wire#powerrail
      Div(in1 := "Settings".OscTorqLimLowPer, in2 := 100.0, out => #TempReal)
      Mul(in1 := #OscTorqRevFtLbs, in2 := #TempReal, out => #OscTorqRevLowLimFtlbs)
      Div(in1 := "Settings".OscTorqLimHighPer, in2 := 100.0, out => #TempReal)
      Mul(in1 := #OscTorqRevFtLbs, in2 := #TempReal, out => #OscTorqRevHighLimFtLbs)
   END_RUNG
   // the same network as SCL:
   #TempReal := #OscSpeedTHper / 100.0;
   #OscSpeedRevZone1 := #TempReal * #OscSpeedRevRPM;
   #TempReal := #TempReal + 0.1;
   #OscSpeedRevZone2 := #TempReal * #OscSpeedRevRPM;
   #TempReal := #OscSpeedHoldper / 100.0;
   #OscSpeedRevZone3 := #TempReal * #OscSpeedRevRPM;
   #TempReal := #TempReal + 0.05;
   #OscSpeedRevZone4 := #TempReal * #OscSpeedRevRPM;
   #TempReal := "Settings".OscTorqLimLowPer / 100.0;
   #OscTorqRevLowLimFtlbs := #OscTorqRevFtLbs * #TempReal;
   #TempReal := "Settings".OscTorqLimHighPer / 100.0;
   #OscTorqRevHighLimFtLbs := #OscTorqRevFtLbs * #TempReal;
END_REGION

REGION Network 12: Visual Oscillator Home Position
   // Set the oscillator home position in relative degrees to be used as the range limit on gauge for home position
   RUNG wire#powerrail
      Add(in1 := #OscHomeRelDeg, in2 := "RotDegPerCount", out => #OscHomeHighRelDeg)
      { S7_Templates := "SrcType := Real" } GT_Contact(in1 := #OscHomeHighRelDeg, in2 := 360.0)
      Sub(in1 := #OscHomeHighRelDeg, in2 := 360.0, out => #OscHomeHighRelDeg)
   END_RUNG
   RUNG wire#powerrail
      Add(in1 := #OscHomeHighRelDeg, in2 := "RotDegPerCount", out => #OscHomeHigh2RelDeg)
      { S7_Templates := "SrcType := Real" } GT_Contact(in1 := #OscHomeHigh2RelDeg, in2 := 360.0)
      Sub(in1 := #OscHomeHigh2RelDeg, in2 := 360.0, out => #OscHomeHigh2RelDeg)
   END_RUNG
   RUNG wire#powerrail
      Sub(in1 := #OscHomeRelDeg, in2 := "RotDegPerCount", out => #OscHomeLowRelDeg)
      { S7_Templates := "SrcType := Real" } LT_Contact(in1 := #OscHomeLowRelDeg, in2 := 0.0)
      Sub(in1 := #OscHomeLowRelDeg, in2 := 360.0, out => #OscHomeLowRelDeg)
   END_RUNG
   RUNG wire#powerrail
      Sub(in1 := #OscHomeLowRelDeg, in2 := "RotDegPerCount", out => #OscHomeLow2RelDeg)
      { S7_Templates := "SrcType := Real" } LT_Contact(in1 := #OscHomeLow2RelDeg, in2 := 0.0)
      Sub(in1 := #OscHomeLow2RelDeg, in2 := 360.0, out => #OscHomeLow2RelDeg)
   END_RUNG
   // the same network as SCL:
   #OscHomeHighRelDeg := #OscHomeRelDeg + "RotDegPerCount";
   IF #OscHomeHighRelDeg > 360.0 THEN #OscHomeHighRelDeg := #OscHomeHighRelDeg - 360.0; END_IF;
   #OscHomeHigh2RelDeg := #OscHomeHighRelDeg + "RotDegPerCount";
   IF #OscHomeHigh2RelDeg > 360.0 THEN #OscHomeHigh2RelDeg := #OscHomeHigh2RelDeg - 360.0; END_IF;
   #OscHomeLowRelDeg := #OscHomeRelDeg - "RotDegPerCount";
   IF #OscHomeLowRelDeg < 0.0 THEN #OscHomeLowRelDeg := #OscHomeLowRelDeg - 360.0; END_IF;
   #OscHomeLow2RelDeg := #OscHomeLowRelDeg - "RotDegPerCount";
   IF #OscHomeLow2RelDeg < 0.0 THEN #OscHomeLow2RelDeg := #OscHomeLow2RelDeg - 360.0; END_IF;
END_REGION

REGION Network 13: Run Lamp Test
   // Turn on the lamp and horn test bits for the set amount of time and reset bit
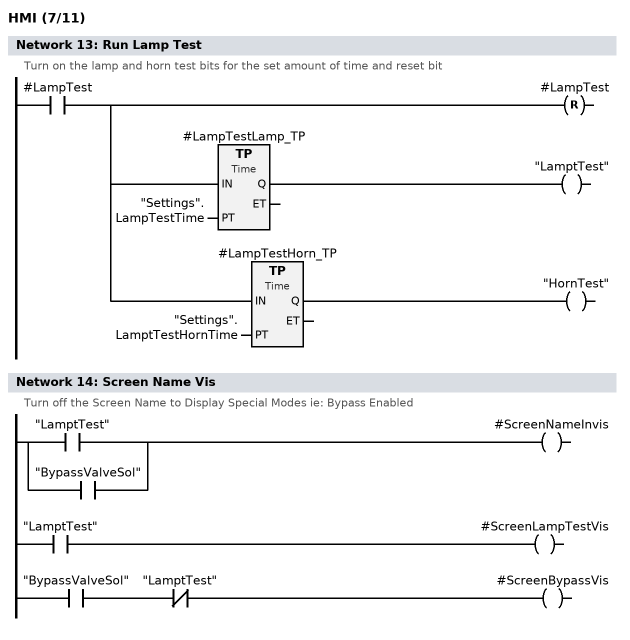
   RUNG wire#powerrail
      Contact( #LampTest )
      wire#w1
      R_Coil( #LampTest )
   END_RUNG
   RUNG wire#w1
      { S7_Templates := "time_type := Time" } #LampTestLamp_TP.TP(pt := "Settings".LampTestTime, et =>)
      Coil( "LamptTest" )
   END_RUNG
   RUNG wire#w1
      { S7_Templates := "time_type := Time" } #LampTestHorn_TP.TP(pt := "Settings".LamptTestHornTime, et =>)
      Coil( "HornTest" )
   END_RUNG
   // the same network as SCL:
   #_w1 := #LampTest;
   IF #_w1 THEN #LampTest := FALSE; END_IF;
   #LampTestLamp_TP(IN := #_w1, PT := "Settings".LampTestTime);   // TP
   "LamptTest" := #LampTestLamp_TP.Q;
   #LampTestHorn_TP(IN := #_w1, PT := "Settings".LamptTestHornTime);   // TP
   "HornTest" := #LampTestHorn_TP.Q;
END_REGION

REGION Network 14: Screen Name Vis
   // Turn off the Screen Name to Display Special Modes ie: Bypass Enabled
   RUNG wire#powerrail
      Contact( "LamptTest" )
      wire#w1
      Coil( #ScreenNameInvis )
   END_RUNG
   RUNG wire#powerrail
      Contact( "BypassValveSol" )
   END_RUNG wire#w1
   RUNG wire#powerrail
      Contact( "LamptTest" )
      Coil( #ScreenLampTestVis )
   END_RUNG
   RUNG wire#powerrail
      Contact( "BypassValveSol" )
      I_Contact( "LamptTest" )
      Coil( #ScreenBypassVis )
   END_RUNG
   // the same network as SCL:
   #ScreenNameInvis := "LamptTest" OR "BypassValveSol";
   #ScreenLampTestVis := "LamptTest";
   #ScreenBypassVis := "BypassValveSol" AND NOT "LamptTest";
END_REGION

REGION Network 15: Oscillator Screen Buttons
   // Set Buttons on based on operations of oscillator
   // Start Button on if Oscillating - State between 200-299
   // Hold Button on if Holding or Bumping - State between 100-199
   // Stop Button on if System Enabled but not Oscillating or Holding/Bumping awaiting Cmd- State 1
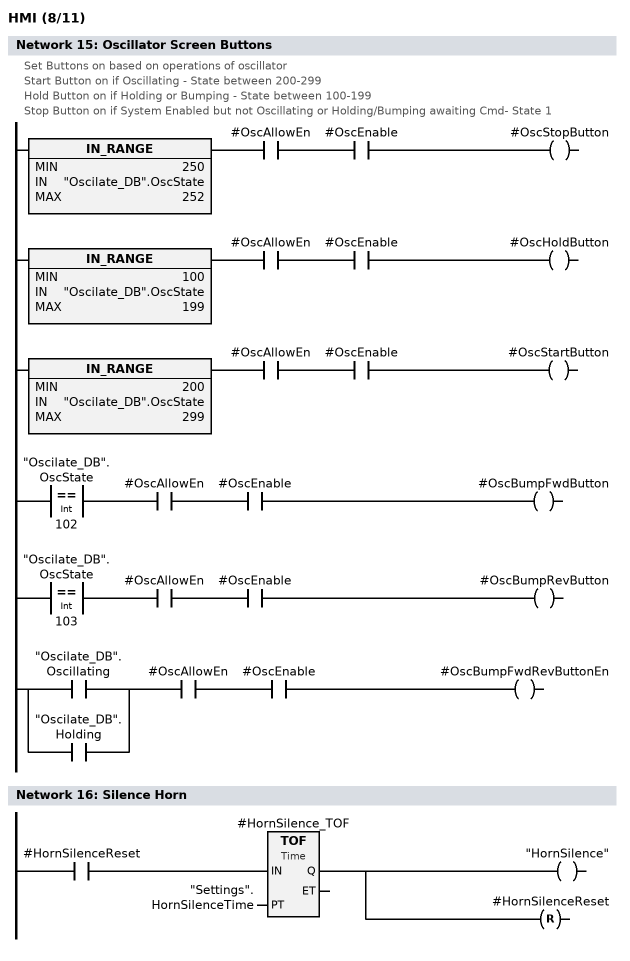
   RUNG wire#powerrail
      { S7_Templates := "SrcType := Int" } InRange(min := 250, in := "Oscilate_DB".OscState, max := 252)
      Contact( #OscAllowEn )
      Contact( #OscEnable )
      Coil( #OscStopButton )
   END_RUNG
   RUNG wire#powerrail
      { S7_Templates := "SrcType := Int" } InRange(min := 100, in := "Oscilate_DB".OscState, max := 199)
      Contact( #OscAllowEn )
      Contact( #OscEnable )
      Coil( #OscHoldButton )
   END_RUNG
   RUNG wire#powerrail
      { S7_Templates := "SrcType := Int" } InRange(min := 200, in := "Oscilate_DB".OscState, max := 299)
      Contact( #OscAllowEn )
      Contact( #OscEnable )
      Coil( #OscStartButton )
   END_RUNG
   RUNG wire#powerrail
      { S7_Templates := "SrcType := Int" } EQ_Contact(in1 := "Oscilate_DB".OscState, in2 := 102)
      Contact( #OscAllowEn )
      Contact( #OscEnable )
      Coil( #OscBumpFwdButton )
   END_RUNG
   RUNG wire#powerrail
      { S7_Templates := "SrcType := Int" } EQ_Contact(in1 := "Oscilate_DB".OscState, in2 := 103)
      Contact( #OscAllowEn )
      Contact( #OscEnable )
      Coil( #OscBumpRevButton )
   END_RUNG
   RUNG wire#powerrail
      Contact( "Oscilate_DB".Oscillating )
      wire#w1
      Contact( #OscAllowEn )
      Contact( #OscEnable )
      Coil( #OscBumpFwdRevButtonEn )
   END_RUNG
   RUNG wire#powerrail
      Contact( "Oscilate_DB".Holding )
   END_RUNG wire#w1
   // the same network as SCL:
   #OscStopButton := (250 <= "Oscilate_DB".OscState) AND ("Oscilate_DB".OscState <= 252) AND #OscAllowEn AND #OscEnable;
   #OscHoldButton := (100 <= "Oscilate_DB".OscState) AND ("Oscilate_DB".OscState <= 199) AND #OscAllowEn AND #OscEnable;
   #OscStartButton := (200 <= "Oscilate_DB".OscState) AND ("Oscilate_DB".OscState <= 299) AND #OscAllowEn AND #OscEnable;
   #OscBumpFwdButton := ("Oscilate_DB".OscState = 102) AND #OscAllowEn AND #OscEnable;
   #OscBumpRevButton := ("Oscilate_DB".OscState = 103) AND #OscAllowEn AND #OscEnable;
   #OscBumpFwdRevButtonEn := ("Oscilate_DB".Oscillating OR "Oscilate_DB".Holding) AND #OscAllowEn AND #OscEnable;
END_REGION

REGION Network 16: Silence Horn
   RUNG wire#powerrail
      Contact( #HornSilenceReset )
      { S7_Templates := "time_type := Time" } #HornSilence_TOF.TOF(pt := "Settings".HornSilenceTime, et =>)
      wire#w1
      Coil( "HornSilence" )
   END_RUNG
   RUNG wire#w1
      R_Coil( #HornSilenceReset )
   END_RUNG
   // the same network as SCL:
   #HornSilence_TOF(IN := #HornSilenceReset, PT := "Settings".HornSilenceTime);   // TOF
   "HornSilence" := #HornSilence_TOF.Q;
   IF #HornSilence_TOF.Q THEN #HornSilenceReset := FALSE; END_IF;
END_REGION

REGION Network 17: Assign Alarms to Alarms1 Int
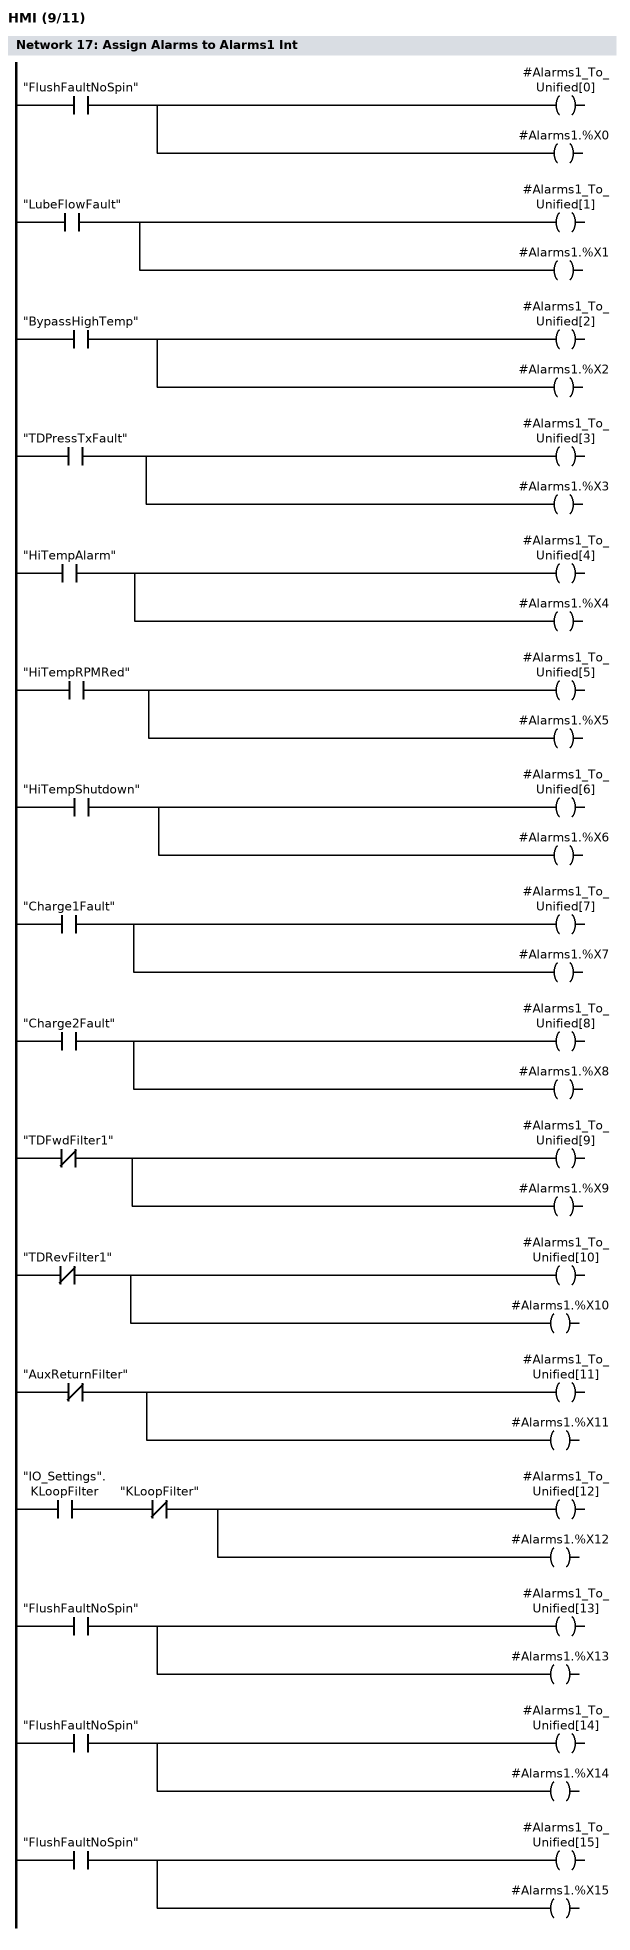
   RUNG wire#powerrail
      Contact( "FlushFaultNoSpin" )
      wire#w1
      Coil( #Alarms1_To_Unified[0] )
   END_RUNG
   RUNG wire#w1
      Coil( #Alarms1.%X0 )
   END_RUNG
   RUNG wire#powerrail
      Contact( "LubeFlowFault" )
      wire#w2
      Coil( #Alarms1_To_Unified[1] )
   END_RUNG
   RUNG wire#w2
      Coil( #Alarms1.%X1 )
   END_RUNG
   RUNG wire#powerrail
      Contact( "BypassHighTemp" )
      wire#w3
      Coil( #Alarms1_To_Unified[2] )
   END_RUNG
   RUNG wire#w3
      Coil( #Alarms1.%X2 )
   END_RUNG
   RUNG wire#powerrail
      Contact( "TDPressTxFault" )
      wire#w4
      Coil( #Alarms1_To_Unified[3] )
   END_RUNG
   RUNG wire#w4
      Coil( #Alarms1.%X3 )
   END_RUNG
   RUNG wire#powerrail
      Contact( "HiTempAlarm" )
      wire#w5
      Coil( #Alarms1_To_Unified[4] )
   END_RUNG
   RUNG wire#w5
      Coil( #Alarms1.%X4 )
   END_RUNG
   RUNG wire#powerrail
      Contact( "HiTempRPMRed" )
      wire#w6
      Coil( #Alarms1_To_Unified[5] )
   END_RUNG
   RUNG wire#w6
      Coil( #Alarms1.%X5 )
   END_RUNG
   RUNG wire#powerrail
      Contact( "HiTempShutdown" )
      wire#w7
      Coil( #Alarms1_To_Unified[6] )
   END_RUNG
   RUNG wire#w7
      Coil( #Alarms1.%X6 )
   END_RUNG
   RUNG wire#powerrail
      Contact( "Charge1Fault" )
      wire#w8
      Coil( #Alarms1_To_Unified[7] )
   END_RUNG
   RUNG wire#w8
      Coil( #Alarms1.%X7 )
   END_RUNG
   RUNG wire#powerrail
      Contact( "Charge2Fault" )
      wire#w9
      Coil( #Alarms1_To_Unified[8] )
   END_RUNG
   RUNG wire#w9
      Coil( #Alarms1.%X8 )
   END_RUNG
   RUNG wire#powerrail
      I_Contact( "TDFwdFilter1" )
      wire#w10
      Coil( #Alarms1_To_Unified[9] )
   END_RUNG
   RUNG wire#w10
      Coil( #Alarms1.%X9 )
   END_RUNG
   RUNG wire#powerrail
      I_Contact( "TDRevFilter1" )
      wire#w11
      Coil( #Alarms1_To_Unified[10] )
   END_RUNG
   RUNG wire#w11
      Coil( #Alarms1.%X10 )
   END_RUNG
   RUNG wire#powerrail
      I_Contact( "AuxReturnFilter" )
      wire#w12
      Coil( #Alarms1_To_Unified[11] )
   END_RUNG
   RUNG wire#w12
      Coil( #Alarms1.%X11 )
   END_RUNG
   RUNG wire#powerrail
      Contact( "IO_Settings".KLoopFilter )
      I_Contact( "KLoopFilter" )
      wire#w13
      Coil( #Alarms1_To_Unified[12] )
   END_RUNG
   RUNG wire#w13
      Coil( #Alarms1.%X12 )
   END_RUNG
   RUNG wire#powerrail
      Contact( "FlushFaultNoSpin" )
      wire#w14
      Coil( #Alarms1_To_Unified[13] )
   END_RUNG
   RUNG wire#w14
      Coil( #Alarms1.%X13 )
   END_RUNG
   RUNG wire#powerrail
      Contact( "FlushFaultNoSpin" )
      wire#w15
      Coil( #Alarms1_To_Unified[14] )
   END_RUNG
   RUNG wire#w15
      Coil( #Alarms1.%X14 )
   END_RUNG
   RUNG wire#powerrail
      Contact( "FlushFaultNoSpin" )
      wire#w16
      Coil( #Alarms1_To_Unified[15] )
   END_RUNG
   RUNG wire#w16
      Coil( #Alarms1.%X15 )
   END_RUNG
   // the same network as SCL:
   #Alarms1_To_Unified[0] := "FlushFaultNoSpin";
   #Alarms1.%X0 := "FlushFaultNoSpin";
   #Alarms1_To_Unified[1] := "LubeFlowFault";
   #Alarms1.%X1 := "LubeFlowFault";
   #Alarms1_To_Unified[2] := "BypassHighTemp";
   #Alarms1.%X2 := "BypassHighTemp";
   #Alarms1_To_Unified[3] := "TDPressTxFault";
   #Alarms1.%X3 := "TDPressTxFault";
   #Alarms1_To_Unified[4] := "HiTempAlarm";
   #Alarms1.%X4 := "HiTempAlarm";
   #Alarms1_To_Unified[5] := "HiTempRPMRed";
   #Alarms1.%X5 := "HiTempRPMRed";
   #Alarms1_To_Unified[6] := "HiTempShutdown";
   #Alarms1.%X6 := "HiTempShutdown";
   #Alarms1_To_Unified[7] := "Charge1Fault";
   #Alarms1.%X7 := "Charge1Fault";
   #Alarms1_To_Unified[8] := "Charge2Fault";
   #Alarms1.%X8 := "Charge2Fault";
   #Alarms1_To_Unified[9] := NOT "TDFwdFilter1";
   #Alarms1.%X9 := NOT "TDFwdFilter1";
   #Alarms1_To_Unified[10] := NOT "TDRevFilter1";
   #Alarms1.%X10 := NOT "TDRevFilter1";
   #Alarms1_To_Unified[11] := NOT "AuxReturnFilter";
   #Alarms1.%X11 := NOT "AuxReturnFilter";
   #Alarms1_To_Unified[12] := "IO_Settings".KLoopFilter AND NOT "KLoopFilter";
   #Alarms1.%X12 := "IO_Settings".KLoopFilter AND NOT "KLoopFilter";
   #Alarms1_To_Unified[13] := "FlushFaultNoSpin";
   #Alarms1.%X13 := "FlushFaultNoSpin";
   #Alarms1_To_Unified[14] := "FlushFaultNoSpin";
   #Alarms1.%X14 := "FlushFaultNoSpin";
   #Alarms1_To_Unified[15] := "FlushFaultNoSpin";
   #Alarms1.%X15 := "FlushFaultNoSpin";
END_REGION

REGION Network 18: Assign Alarms to Alarms2 Int
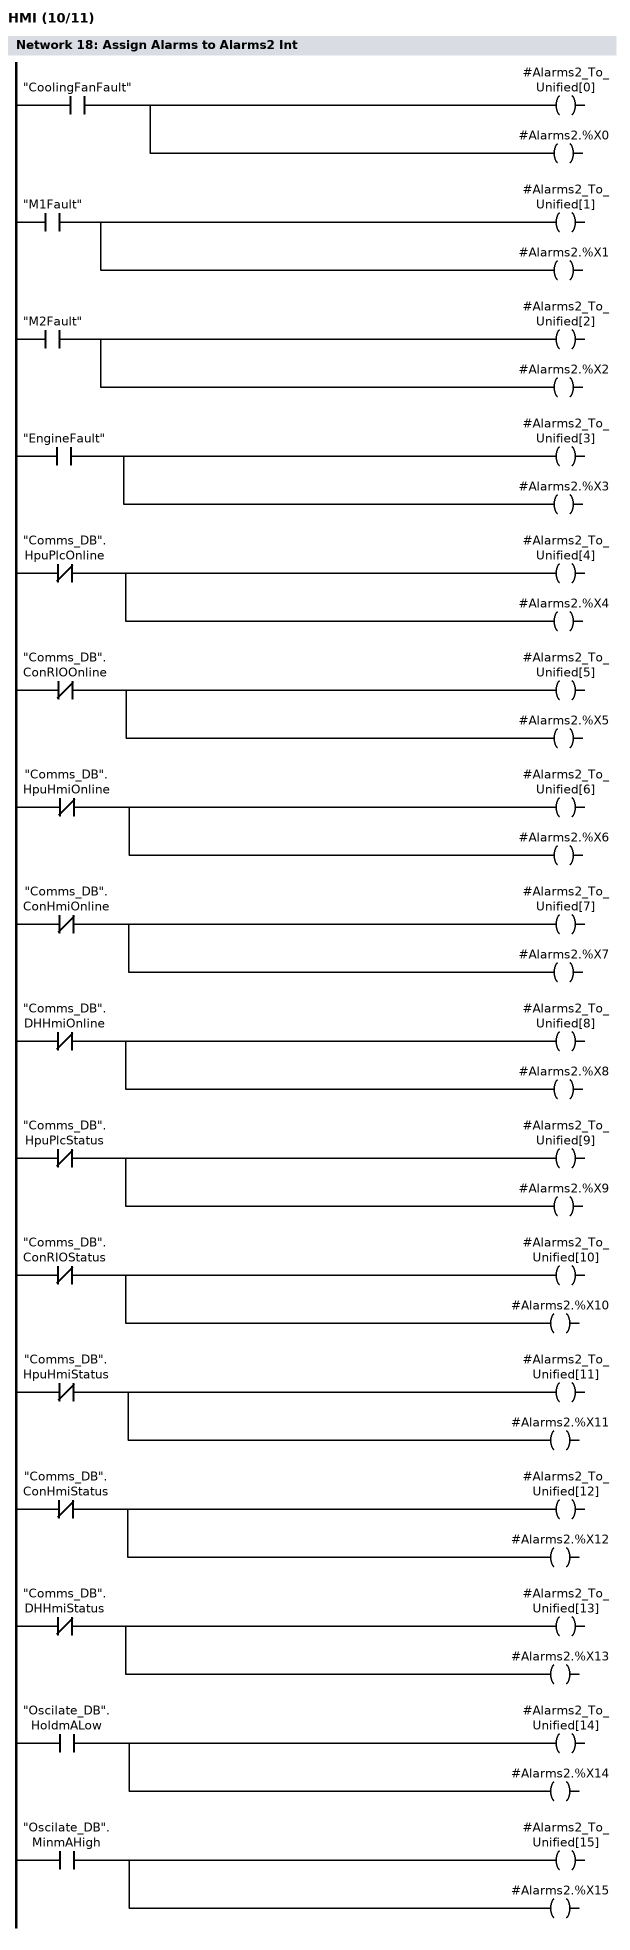
   RUNG wire#powerrail
      Contact( "CoolingFanFault" )
      wire#w1
      Coil( #Alarms2_To_Unified[0] )
   END_RUNG
   RUNG wire#w1
      Coil( #Alarms2.%X0 )
   END_RUNG
   RUNG wire#powerrail
      Contact( "M1Fault" )
      wire#w2
      Coil( #Alarms2_To_Unified[1] )
   END_RUNG
   RUNG wire#w2
      Coil( #Alarms2.%X1 )
   END_RUNG
   RUNG wire#powerrail
      Contact( "M2Fault" )
      wire#w3
      Coil( #Alarms2_To_Unified[2] )
   END_RUNG
   RUNG wire#w3
      Coil( #Alarms2.%X2 )
   END_RUNG
   RUNG wire#powerrail
      Contact( "EngineFault" )
      wire#w4
      Coil( #Alarms2_To_Unified[3] )
   END_RUNG
   RUNG wire#w4
      Coil( #Alarms2.%X3 )
   END_RUNG
   RUNG wire#powerrail
      I_Contact( "Comms_DB".HpuPlcOnline )
      wire#w5
      Coil( #Alarms2_To_Unified[4] )
   END_RUNG
   RUNG wire#w5
      Coil( #Alarms2.%X4 )
   END_RUNG
   RUNG wire#powerrail
      I_Contact( "Comms_DB".ConRIOOnline )
      wire#w6
      Coil( #Alarms2_To_Unified[5] )
   END_RUNG
   RUNG wire#w6
      Coil( #Alarms2.%X5 )
   END_RUNG
   RUNG wire#powerrail
      I_Contact( "Comms_DB".HpuHmiOnline )
      wire#w7
      Coil( #Alarms2_To_Unified[6] )
   END_RUNG
   RUNG wire#w7
      Coil( #Alarms2.%X6 )
   END_RUNG
   RUNG wire#powerrail
      I_Contact( "Comms_DB".ConHmiOnline )
      wire#w8
      Coil( #Alarms2_To_Unified[7] )
   END_RUNG
   RUNG wire#w8
      Coil( #Alarms2.%X7 )
   END_RUNG
   RUNG wire#powerrail
      I_Contact( "Comms_DB".DHHmiOnline )
      wire#w9
      Coil( #Alarms2_To_Unified[8] )
   END_RUNG
   RUNG wire#w9
      Coil( #Alarms2.%X8 )
   END_RUNG
   RUNG wire#powerrail
      I_Contact( "Comms_DB".HpuPlcStatus )
      wire#w10
      Coil( #Alarms2_To_Unified[9] )
   END_RUNG
   RUNG wire#w10
      Coil( #Alarms2.%X9 )
   END_RUNG
   RUNG wire#powerrail
      I_Contact( "Comms_DB".ConRIOStatus )
      wire#w11
      Coil( #Alarms2_To_Unified[10] )
   END_RUNG
   RUNG wire#w11
      Coil( #Alarms2.%X10 )
   END_RUNG
   RUNG wire#powerrail
      I_Contact( "Comms_DB".HpuHmiStatus )
      wire#w12
      Coil( #Alarms2_To_Unified[11] )
   END_RUNG
   RUNG wire#w12
      Coil( #Alarms2.%X11 )
   END_RUNG
   RUNG wire#powerrail
      I_Contact( "Comms_DB".ConHmiStatus )
      wire#w13
      Coil( #Alarms2_To_Unified[12] )
   END_RUNG
   RUNG wire#w13
      Coil( #Alarms2.%X12 )
   END_RUNG
   RUNG wire#powerrail
      I_Contact( "Comms_DB".DHHmiStatus )
      wire#w14
      Coil( #Alarms2_To_Unified[13] )
   END_RUNG
   RUNG wire#w14
      Coil( #Alarms2.%X13 )
   END_RUNG
   RUNG wire#powerrail
      Contact( "Oscilate_DB".HoldmALow )
      wire#w15
      Coil( #Alarms2_To_Unified[14] )
   END_RUNG
   RUNG wire#w15
      Coil( #Alarms2.%X14 )
   END_RUNG
   RUNG wire#powerrail
      Contact( "Oscilate_DB".MinmAHigh )
      wire#w16
      Coil( #Alarms2_To_Unified[15] )
   END_RUNG
   RUNG wire#w16
      Coil( #Alarms2.%X15 )
   END_RUNG
   // the same network as SCL:
   #Alarms2_To_Unified[0] := "CoolingFanFault";
   #Alarms2.%X0 := "CoolingFanFault";
   #Alarms2_To_Unified[1] := "M1Fault";
   #Alarms2.%X1 := "M1Fault";
   #Alarms2_To_Unified[2] := "M2Fault";
   #Alarms2.%X2 := "M2Fault";
   #Alarms2_To_Unified[3] := "EngineFault";
   #Alarms2.%X3 := "EngineFault";
   #Alarms2_To_Unified[4] := NOT "Comms_DB".HpuPlcOnline;
   #Alarms2.%X4 := NOT "Comms_DB".HpuPlcOnline;
   #Alarms2_To_Unified[5] := NOT "Comms_DB".ConRIOOnline;
   #Alarms2.%X5 := NOT "Comms_DB".ConRIOOnline;
   #Alarms2_To_Unified[6] := NOT "Comms_DB".HpuHmiOnline;
   #Alarms2.%X6 := NOT "Comms_DB".HpuHmiOnline;
   #Alarms2_To_Unified[7] := NOT "Comms_DB".ConHmiOnline;
   #Alarms2.%X7 := NOT "Comms_DB".ConHmiOnline;
   #Alarms2_To_Unified[8] := NOT "Comms_DB".DHHmiOnline;
   #Alarms2.%X8 := NOT "Comms_DB".DHHmiOnline;
   #Alarms2_To_Unified[9] := NOT "Comms_DB".HpuPlcStatus;
   #Alarms2.%X9 := NOT "Comms_DB".HpuPlcStatus;
   #Alarms2_To_Unified[10] := NOT "Comms_DB".ConRIOStatus;
   #Alarms2.%X10 := NOT "Comms_DB".ConRIOStatus;
   #Alarms2_To_Unified[11] := NOT "Comms_DB".HpuHmiStatus;
   #Alarms2.%X11 := NOT "Comms_DB".HpuHmiStatus;
   #Alarms2_To_Unified[12] := NOT "Comms_DB".ConHmiStatus;
   #Alarms2.%X12 := NOT "Comms_DB".ConHmiStatus;
   #Alarms2_To_Unified[13] := NOT "Comms_DB".DHHmiStatus;
   #Alarms2.%X13 := NOT "Comms_DB".DHHmiStatus;
   #Alarms2_To_Unified[14] := "Oscilate_DB".HoldmALow;
   #Alarms2.%X14 := "Oscilate_DB".HoldmALow;
   #Alarms2_To_Unified[15] := "Oscilate_DB".MinmAHigh;
   #Alarms2.%X15 := "Oscilate_DB".MinmAHigh;
END_REGION

REGION Network 19: Assign Warnings to Warnings Int
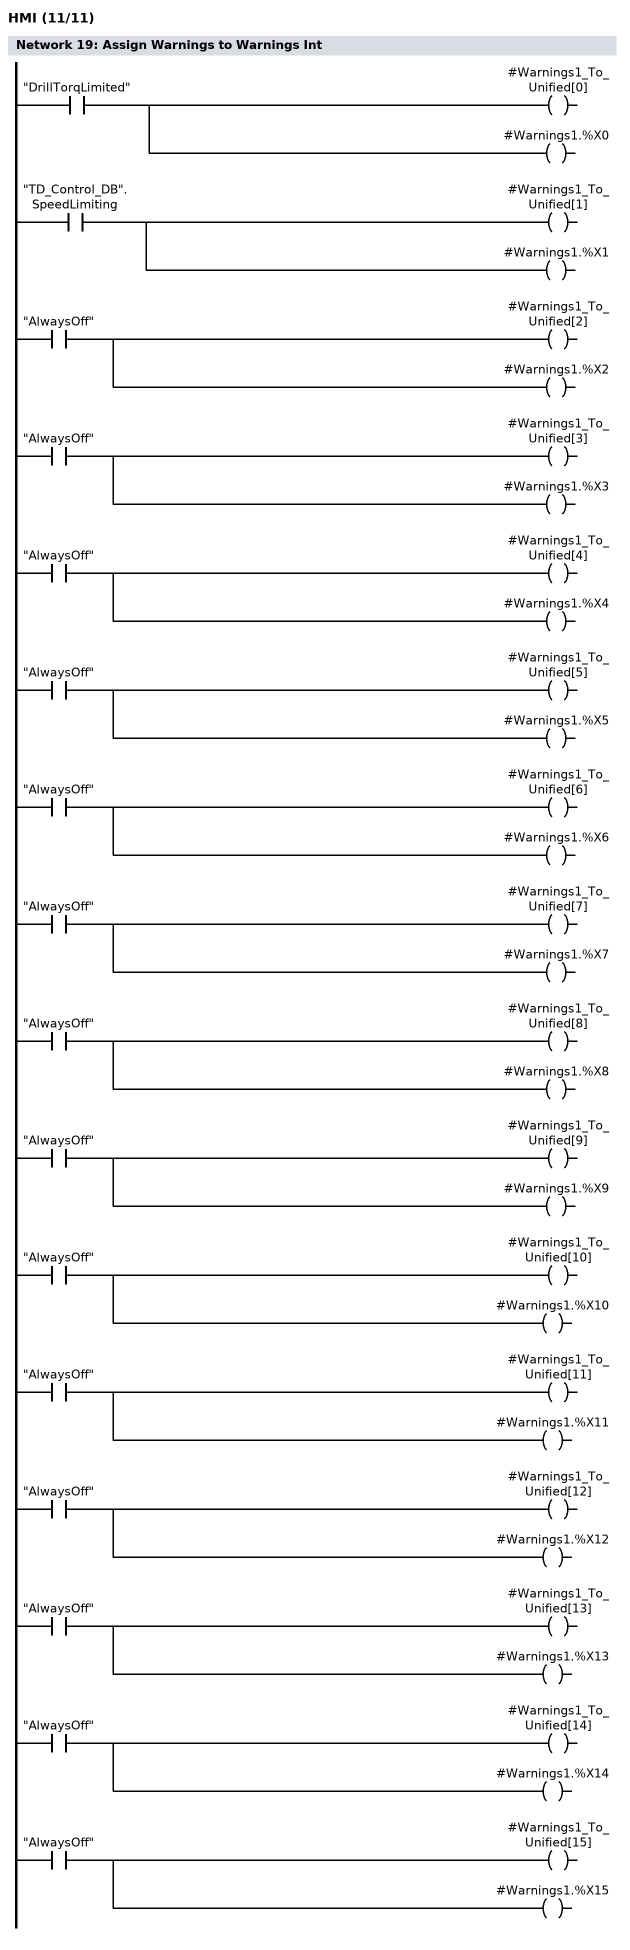
   RUNG wire#powerrail
      Contact( "DrillTorqLimited" )
      wire#w1
      Coil( #Warnings1_To_Unified[0] )
   END_RUNG
   RUNG wire#w1
      Coil( #Warnings1.%X0 )
   END_RUNG
   RUNG wire#powerrail
      Contact( "TD_Control_DB".SpeedLimiting )
      wire#w2
      Coil( #Warnings1_To_Unified[1] )
   END_RUNG
   RUNG wire#w2
      Coil( #Warnings1.%X1 )
   END_RUNG
   RUNG wire#powerrail
      Contact( "AlwaysOff" )
      wire#w3
      Coil( #Warnings1_To_Unified[2] )
   END_RUNG
   RUNG wire#w3
      Coil( #Warnings1.%X2 )
   END_RUNG
   RUNG wire#powerrail
      Contact( "AlwaysOff" )
      wire#w4
      Coil( #Warnings1_To_Unified[3] )
   END_RUNG
   RUNG wire#w4
      Coil( #Warnings1.%X3 )
   END_RUNG
   RUNG wire#powerrail
      Contact( "AlwaysOff" )
      wire#w5
      Coil( #Warnings1_To_Unified[4] )
   END_RUNG
   RUNG wire#w5
      Coil( #Warnings1.%X4 )
   END_RUNG
   RUNG wire#powerrail
      Contact( "AlwaysOff" )
      wire#w6
      Coil( #Warnings1_To_Unified[5] )
   END_RUNG
   RUNG wire#w6
      Coil( #Warnings1.%X5 )
   END_RUNG
   RUNG wire#powerrail
      Contact( "AlwaysOff" )
      wire#w7
      Coil( #Warnings1_To_Unified[6] )
   END_RUNG
   RUNG wire#w7
      Coil( #Warnings1.%X6 )
   END_RUNG
   RUNG wire#powerrail
      Contact( "AlwaysOff" )
      wire#w8
      Coil( #Warnings1_To_Unified[7] )
   END_RUNG
   RUNG wire#w8
      Coil( #Warnings1.%X7 )
   END_RUNG
   RUNG wire#powerrail
      Contact( "AlwaysOff" )
      wire#w9
      Coil( #Warnings1_To_Unified[8] )
   END_RUNG
   RUNG wire#w9
      Coil( #Warnings1.%X8 )
   END_RUNG
   RUNG wire#powerrail
      Contact( "AlwaysOff" )
      wire#w10
      Coil( #Warnings1_To_Unified[9] )
   END_RUNG
   RUNG wire#w10
      Coil( #Warnings1.%X9 )
   END_RUNG
   RUNG wire#powerrail
      Contact( "AlwaysOff" )
      wire#w11
      Coil( #Warnings1_To_Unified[10] )
   END_RUNG
   RUNG wire#w11
      Coil( #Warnings1.%X10 )
   END_RUNG
   RUNG wire#powerrail
      Contact( "AlwaysOff" )
      wire#w12
      Coil( #Warnings1_To_Unified[11] )
   END_RUNG
   RUNG wire#w12
      Coil( #Warnings1.%X11 )
   END_RUNG
   RUNG wire#powerrail
      Contact( "AlwaysOff" )
      wire#w13
      Coil( #Warnings1_To_Unified[12] )
   END_RUNG
   RUNG wire#w13
      Coil( #Warnings1.%X12 )
   END_RUNG
   RUNG wire#powerrail
      Contact( "AlwaysOff" )
      wire#w14
      Coil( #Warnings1_To_Unified[13] )
   END_RUNG
   RUNG wire#w14
      Coil( #Warnings1.%X13 )
   END_RUNG
   RUNG wire#powerrail
      Contact( "AlwaysOff" )
      wire#w15
      Coil( #Warnings1_To_Unified[14] )
   END_RUNG
   RUNG wire#w15
      Coil( #Warnings1.%X14 )
   END_RUNG
   RUNG wire#powerrail
      Contact( "AlwaysOff" )
      wire#w16
      Coil( #Warnings1_To_Unified[15] )
   END_RUNG
   RUNG wire#w16
      Coil( #Warnings1.%X15 )
   END_RUNG
   // the same network as SCL:
   #Warnings1_To_Unified[0] := "DrillTorqLimited";
   #Warnings1.%X0 := "DrillTorqLimited";
   #Warnings1_To_Unified[1] := "TD_Control_DB".SpeedLimiting;
   #Warnings1.%X1 := "TD_Control_DB".SpeedLimiting;
   #Warnings1_To_Unified[2] := "AlwaysOff";
   #Warnings1.%X2 := "AlwaysOff";
   #Warnings1_To_Unified[3] := "AlwaysOff";
   #Warnings1.%X3 := "AlwaysOff";
   #Warnings1_To_Unified[4] := "AlwaysOff";
   #Warnings1.%X4 := "AlwaysOff";
   #Warnings1_To_Unified[5] := "AlwaysOff";
   #Warnings1.%X5 := "AlwaysOff";
   #Warnings1_To_Unified[6] := "AlwaysOff";
   #Warnings1.%X6 := "AlwaysOff";
   #Warnings1_To_Unified[7] := "AlwaysOff";
   #Warnings1.%X7 := "AlwaysOff";
   #Warnings1_To_Unified[8] := "AlwaysOff";
   #Warnings1.%X8 := "AlwaysOff";
   #Warnings1_To_Unified[9] := "AlwaysOff";
   #Warnings1.%X9 := "AlwaysOff";
   #Warnings1_To_Unified[10] := "AlwaysOff";
   #Warnings1.%X10 := "AlwaysOff";
   #Warnings1_To_Unified[11] := "AlwaysOff";
   #Warnings1.%X11 := "AlwaysOff";
   #Warnings1_To_Unified[12] := "AlwaysOff";
   #Warnings1.%X12 := "AlwaysOff";
   #Warnings1_To_Unified[13] := "AlwaysOff";
   #Warnings1.%X13 := "AlwaysOff";
   #Warnings1_To_Unified[14] := "AlwaysOff";
   #Warnings1.%X14 := "AlwaysOff";
   #Warnings1_To_Unified[15] := "AlwaysOff";
   #Warnings1.%X15 := "AlwaysOff";
END_REGION
END_FUNCTION_BLOCK
